(* Logix 5000 project; controller NSH_PLC1 vendor 1 type 14 code 167 rev 32.11; software revision 32.02; part 6 of 12 *)
(* tags used below, declared in another part *)
   HS_AlarmPulseHorn : BOOL;   // Huller Sheller, New Alarm, Pulse Horn
   HS_FaultResetHorn : BOOL;   // Hullwe Sheller, Fault Reset, sound Horn
   Num_Faults : DINT;   // Number of Huller-Sheller Faults
   Num_Warnings : DINT;   // Number of Huller-Sheller Warnings
   TempMotor : Motor;   // Temp Motor Tag for Subroutines
   BH1 : Motor;   // Auger
   BH1A : Motor;   // Fan
   BH1B : Motor;   // Rev.Fan
   BH1C : Motor;   // Rev. Arm
   BH1D : Motor;   // Airlock
   BH2 : Motor;   // S. Ele
   BH2A : Motor;   // Fan
   BH2B : Motor;   // Rev.Fan
   BH2C : Motor;   // Rev. Arm
   BH2D : Motor;   // Airlock
   BH3A : Motor;   // Fan
   BH3B : Motor;   // Rev.Fan
   BH3C : Motor;   // Rev. Arm
   BH3D : Motor;   // Airlock
   C1A : Motor;   // Auger
   C1B : Motor;   // Auger
   C2 : Motor;   // Auger
   C3A : Motor;   // Auger
   C3B : Motor;   // Auger
   C4 : Motor;   // Ele.
   C7 : Motor;   // Ele
   CR_LastBH1Fan : BOOL;   // Last Motor in Baghouse 1 Fans Running
   CR_RunBH_Fans : BOOL;   // Run Baghouse's Fans Relay
   CR_RunBH_FansCO : BOOL;   // Run Baghouse's Cleanout Relay
   CR_RunHS : BOOL;   // Run Hullers & Shellers Relay
   CR_RunPC1_Fans : BOOL;   // Pre Clean Run Line 1 Fans Relay
   CR_StopHS : BOOL;   // Stop Hullers & Shellers Relay
   D10 : Motor;   // Ele
   D1A : Motor;   // Auger
   D1B : Motor;   // Auger
   D2 : Motor;   // Auger
   D4 : Motor;   // Auger
   D5 : Motor;   // Auger
   D6 : Motor;   // Auger
   H1 : Motor;   // Conv.
   H11 : Motor;   // Ele.
   H12 : Motor;   // Auger
   H13 : Motor;   // Auger
   H14A : Motor;   // Shr. Roll
   H14B : Motor;   // Shr. Roll
   H14C : Motor;   // Vib.
   H16 : Motor;   // Auger
   H17 : Motor;   // Roll Fd.
   H18A : Motor;   // Shr. Roll
   H18B : Motor;   // Shr. Roll
   H18C : Motor;   // Vib.
   H19A : Motor;   // Aspirator
   H19B : Motor;   // Aspirator
   H22 : Motor;   // BMM
   H23A : Motor;   // Aspirator
   H23B : Motor;   // Aspirator
   H24A : Motor;   // Aspirator
   H24B : Motor;   // Aspirator
   H3A : Motor;   // Incline
   H3B : Motor;   // Ele.
   H4 : Motor;   // Auger
   H5 : Motor;   // Auger
   H6 : Motor;   // Roll Fd.
   H7 : Motor;   // BMM
   H8A : Motor;   // Aspirator
   H8B : Motor;   // Aspirator
   H9A : Motor;   // Aspirator
   H9B : Motor;   // Aspirator
   HS_Horn : BOOL;   // Huller Sheller, Horn Output
   HS_LastMotor : BOOL;   // Last Motor in Huller Sheller Sequence is Running
   HS_Starting : BOOL;   // Sheller Sequence is Starting, Prevent Preclean from Starting
   M12aA : Motor;   // Grav.Sep
   M12aB : Motor;   // Syntron
   M13aA : Motor;   // Grav.Sep
   M13aB : Motor;   // Syntron
   M14 : Motor;   // Vib.
   M15 : Motor;   // Ele.
   M16R : Motor;   // Conveyor
   M20 : Motor;   // Ele.
   M21 : Motor;   // Nolin
   M25 : Motor;   // Accept Vib.
   M33 : Motor;   // Belt
   M34 : Motor;   // Destoner
   M35 : Motor;   // Ele.
   M36A : Motor;   // G. Sep.
   M36B : Motor;   // R. Feeder.
   M42C : Motor;   // 3C Deck
   M42D : Motor;   // 3C Deck
   M43CA : Motor;   // Asp.
   M43CB : Motor;   // Asp.
   M43DA : Motor;   // Asp.
   M43DB : Motor;   // Asp.
   P2B : Motor;   // Stick Reel
   PB_HS_Inshell : BOOL;   // Hullers & Shellers Run Inshell Button
   PB_HS_Meats : BOOL;   // Hullers & Shellers Run Meats Button
   PB_StartHS : BOOL;   // Start Hullers & Shellers Button
   PB_StartPC1_Fans : BOOL;   // Pre Clean Start Line 1 Fans Button
   PB_StopHS : BOOL;   // Stop Hullers & Shellers Button
   PBB1D : Motor;   // Fan,
   PBL_HS_Inshell : BOOL;   // Hullers & Shellers Run Inshell Button Light
   PBL_HS_Meats : BOOL;   // Hullers & Shellers Run Meats Button Light
   PBL_StartHS : BOOL;   // Start Hullers & Shellers Button Light
   PBL_StopHS : BOOL;   // Stop Hullers & Shellers Button Light
   PC_FansStarting : BOOL;   // Pre Clean Fans Starting
   PC_LinesStarting : BOOL;   // Pre Clean Line 1 or 2 Starting
   PC_NoEstops : BOOL;   // PreClean, No Estops
   S11 : Motor;   // Ele.
   S12 : Motor;   // Auger
   T1 : Motor;   // Belt
   T2 : Motor;   // Belt
   T3 : Motor;   // Belt
   TMR_StartBH_Fans : TIMER;   // Start Baghouse's Fans Timer
   TMR_StartBH_FansCO : TIMER;   // Start Baghouse's Cleanout Timer
   TMR_StartHS : TIMER;   // Run Hullers & Shellers Warning Timer
(* HullerSheller, continued *)

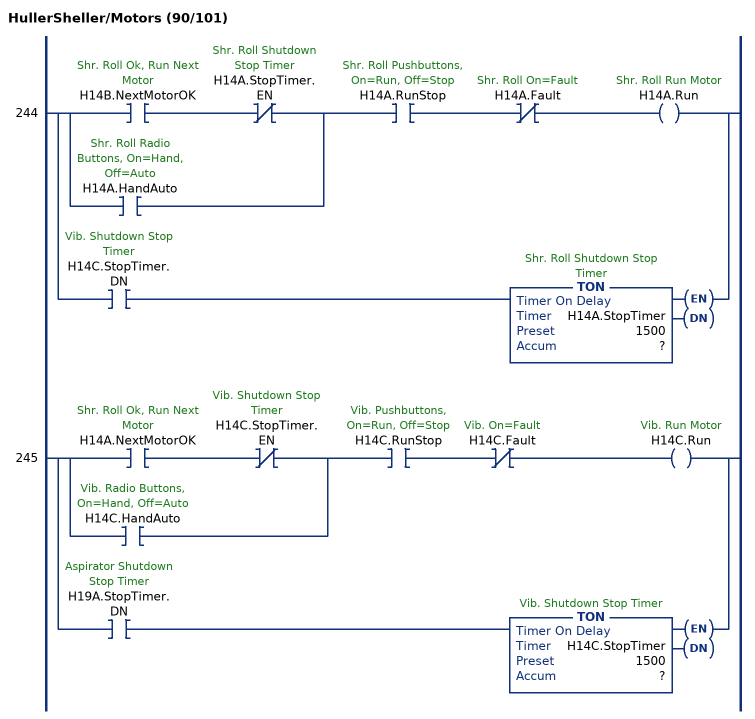
   244: [[XIC(H14B.NextMotorOK) XIO(H14A.StopTimer.EN) ,XIC(H14A.HandAuto) ] XIC(H14A.RunStop) XIO(H14A.Fault) OTE(H14A.Run) ,XIC(H14C.StopTimer.DN) TON(H14A.StopTimer,?,?) ];
   245: [[XIC(H14A.NextMotorOK) XIO(H14C.StopTimer.EN) ,XIC(H14C.HandAuto) ] XIC(H14C.RunStop) XIO(H14C.Fault) OTE(H14C.Run) ,XIC(H19A.StopTimer.DN) TON(H14C.StopTimer,?,?) ];
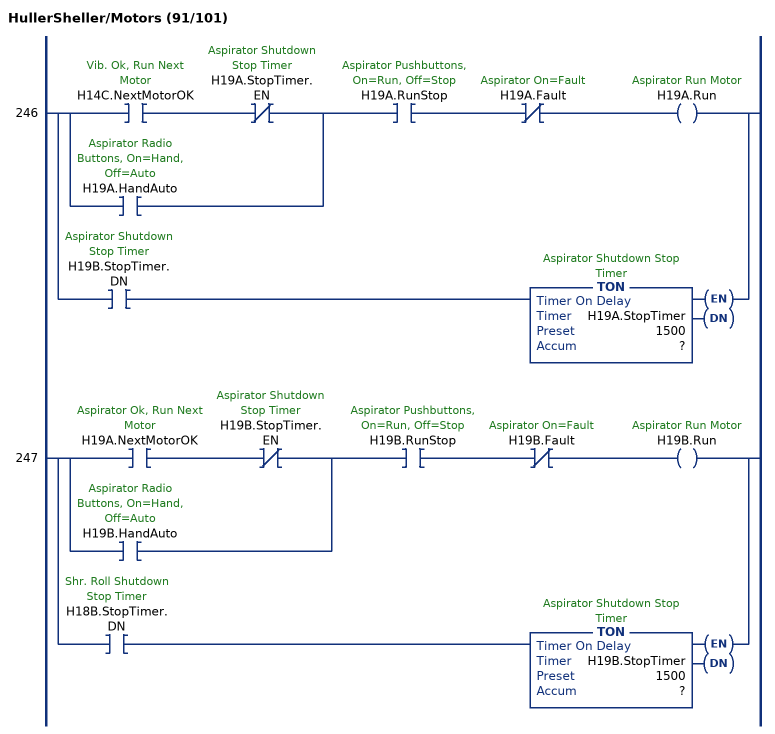
   246: [[XIC(H14C.NextMotorOK) XIO(H19A.StopTimer.EN) ,XIC(H19A.HandAuto) ] XIC(H19A.RunStop) XIO(H19A.Fault) OTE(H19A.Run) ,XIC(H19B.StopTimer.DN) TON(H19A.StopTimer,?,?) ];
   247: [[XIC(H19A.NextMotorOK) XIO(H19B.StopTimer.EN) ,XIC(H19B.HandAuto) ] XIC(H19B.RunStop) XIO(H19B.Fault) OTE(H19B.Run) ,XIC(H18B.StopTimer.DN) TON(H19B.StopTimer,?,?) ];
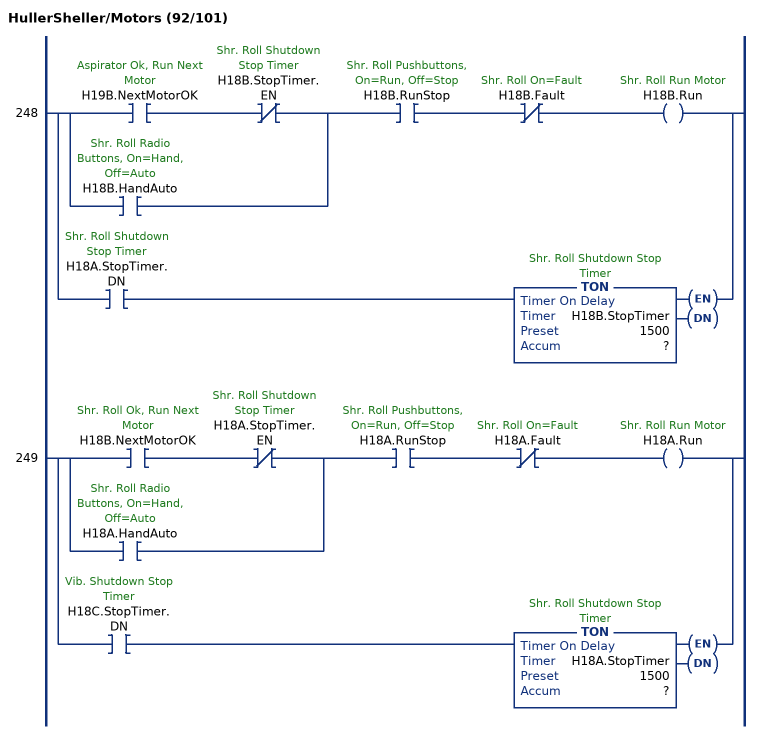
   248: [[XIC(H19B.NextMotorOK) XIO(H18B.StopTimer.EN) ,XIC(H18B.HandAuto) ] XIC(H18B.RunStop) XIO(H18B.Fault) OTE(H18B.Run) ,XIC(H18A.StopTimer.DN) TON(H18B.StopTimer,?,?) ];
   249: [[XIC(H18B.NextMotorOK) XIO(H18A.StopTimer.EN) ,XIC(H18A.HandAuto) ] XIC(H18A.RunStop) XIO(H18A.Fault) OTE(H18A.Run) ,XIC(H18C.StopTimer.DN) TON(H18A.StopTimer,?,?) ];
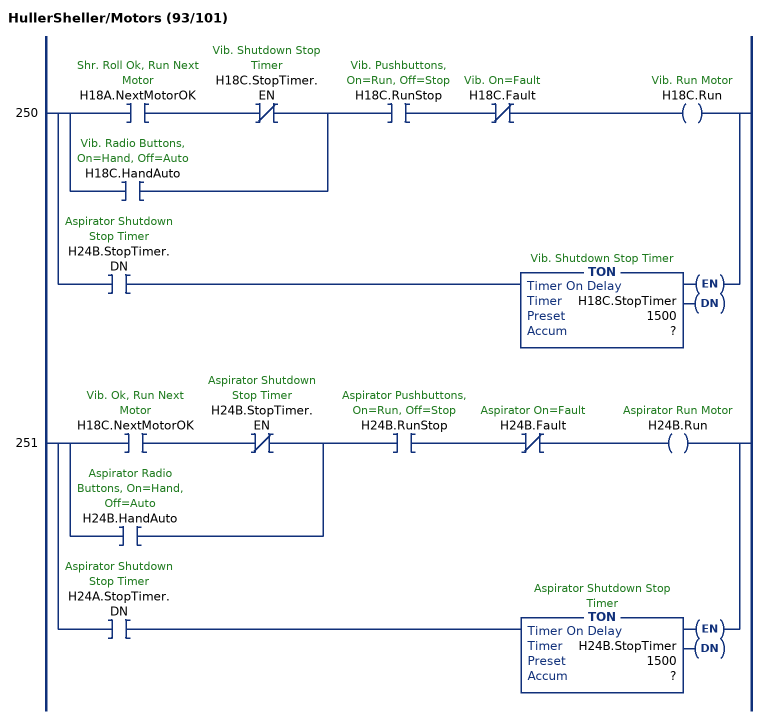
   250: [[XIC(H18A.NextMotorOK) XIO(H18C.StopTimer.EN) ,XIC(H18C.HandAuto) ] XIC(H18C.RunStop) XIO(H18C.Fault) OTE(H18C.Run) ,XIC(H24B.StopTimer.DN) TON(H18C.StopTimer,?,?) ];
   251: [[XIC(H18C.NextMotorOK) XIO(H24B.StopTimer.EN) ,XIC(H24B.HandAuto) ] XIC(H24B.RunStop) XIO(H24B.Fault) OTE(H24B.Run) ,XIC(H24A.StopTimer.DN) TON(H24B.StopTimer,?,?) ];
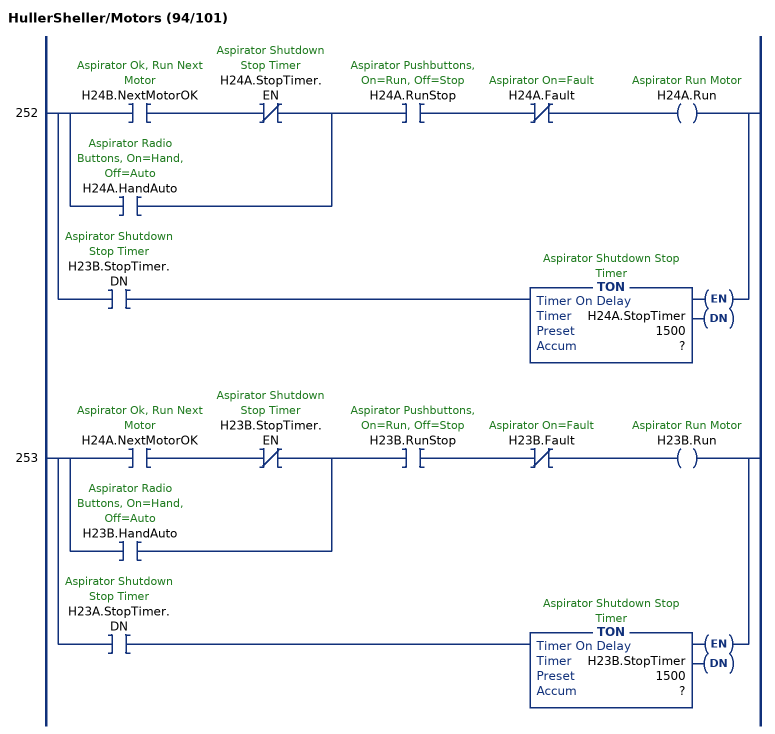
   252: [[XIC(H24B.NextMotorOK) XIO(H24A.StopTimer.EN) ,XIC(H24A.HandAuto) ] XIC(H24A.RunStop) XIO(H24A.Fault) OTE(H24A.Run) ,XIC(H23B.StopTimer.DN) TON(H24A.StopTimer,?,?) ];
   253: [[XIC(H24A.NextMotorOK) XIO(H23B.StopTimer.EN) ,XIC(H23B.HandAuto) ] XIC(H23B.RunStop) XIO(H23B.Fault) OTE(H23B.Run) ,XIC(H23A.StopTimer.DN) TON(H23B.StopTimer,?,?) ];
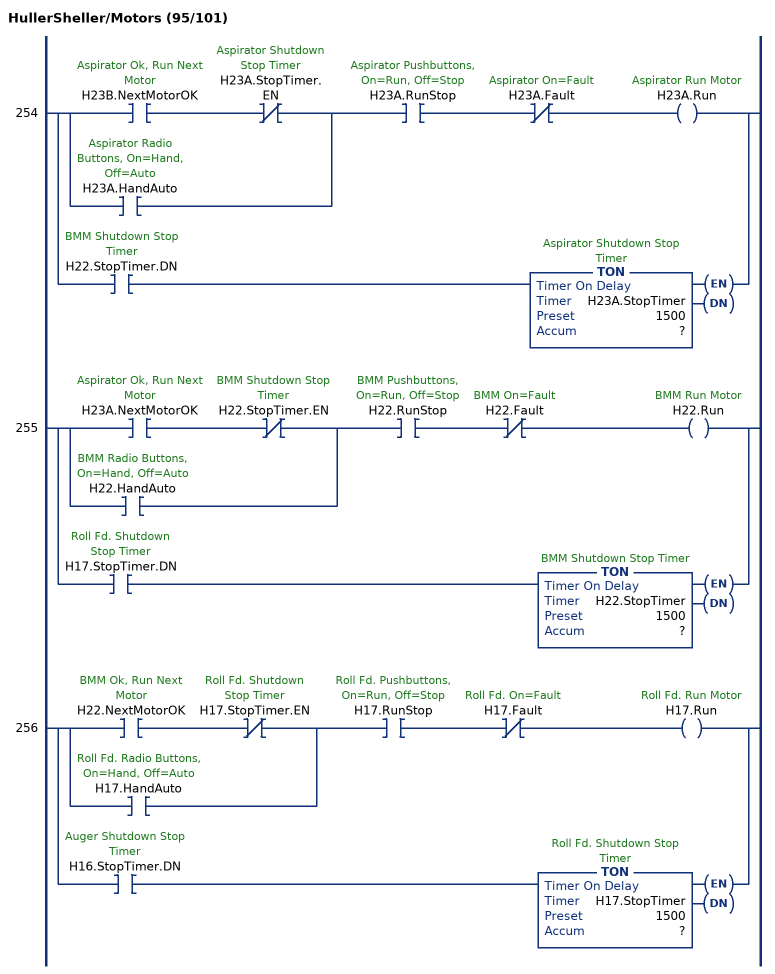
   254: [[XIC(H23B.NextMotorOK) XIO(H23A.StopTimer.EN) ,XIC(H23A.HandAuto) ] XIC(H23A.RunStop) XIO(H23A.Fault) OTE(H23A.Run) ,XIC(H22.StopTimer.DN) TON(H23A.StopTimer,?,?) ];
   255: [[XIC(H23A.NextMotorOK) XIO(H22.StopTimer.EN) ,XIC(H22.HandAuto) ] XIC(H22.RunStop) XIO(H22.Fault) OTE(H22.Run) ,XIC(H17.StopTimer.DN) TON(H22.StopTimer,?,?) ];
   256: [[XIC(H22.NextMotorOK) XIO(H17.StopTimer.EN) ,XIC(H17.HandAuto) ] XIC(H17.RunStop) XIO(H17.Fault) OTE(H17.Run) ,XIC(H16.StopTimer.DN) TON(H17.StopTimer,?,?) ];
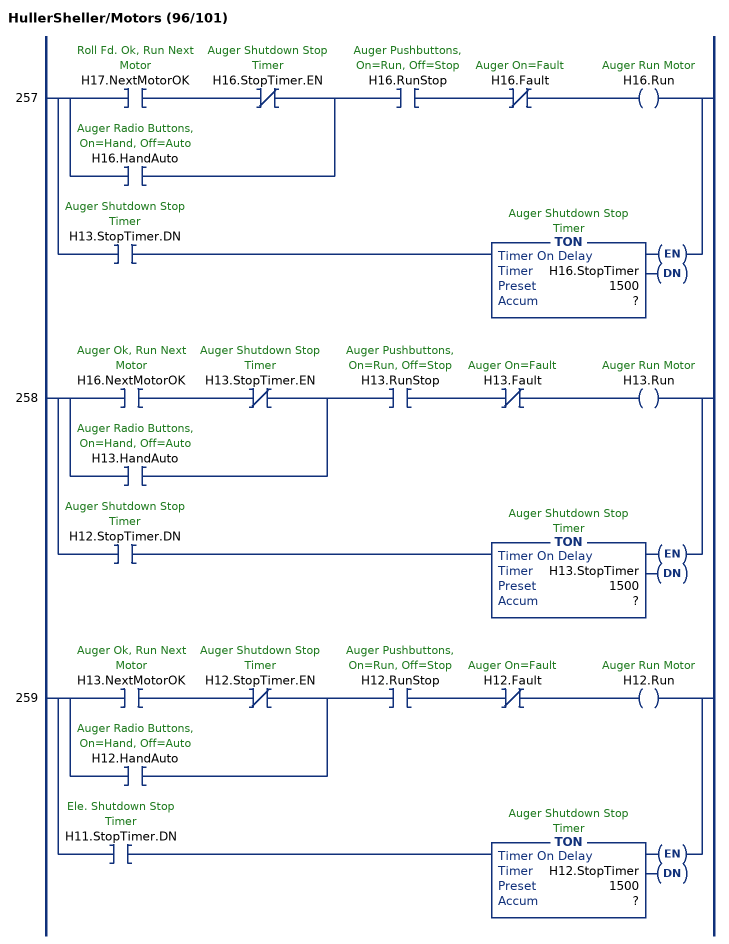
   257: [[XIC(H17.NextMotorOK) XIO(H16.StopTimer.EN) ,XIC(H16.HandAuto) ] XIC(H16.RunStop) XIO(H16.Fault) OTE(H16.Run) ,XIC(H13.StopTimer.DN) TON(H16.StopTimer,?,?) ];
   258: [[XIC(H16.NextMotorOK) XIO(H13.StopTimer.EN) ,XIC(H13.HandAuto) ] XIC(H13.RunStop) XIO(H13.Fault) OTE(H13.Run) ,XIC(H12.StopTimer.DN) TON(H13.StopTimer,?,?) ];
   259: [[XIC(H13.NextMotorOK) XIO(H12.StopTimer.EN) ,XIC(H12.HandAuto) ] XIC(H12.RunStop) XIO(H12.Fault) OTE(H12.Run) ,XIC(H11.StopTimer.DN) TON(H12.StopTimer,?,?) ];
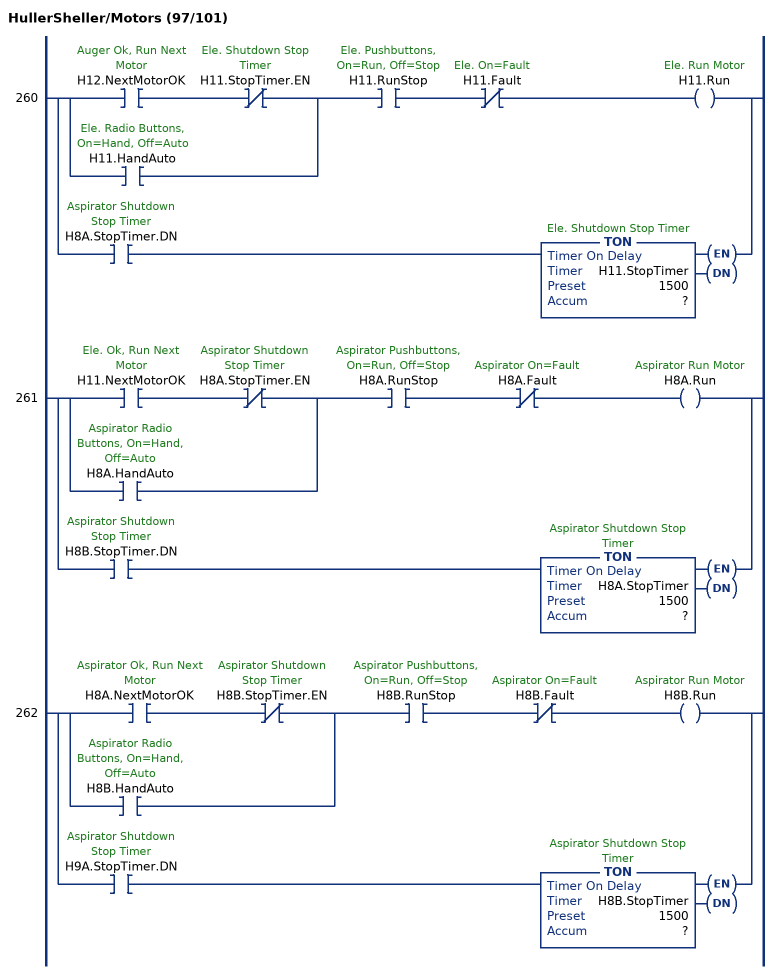
   260: [[XIC(H12.NextMotorOK) XIO(H11.StopTimer.EN) ,XIC(H11.HandAuto) ] XIC(H11.RunStop) XIO(H11.Fault) OTE(H11.Run) ,XIC(H8A.StopTimer.DN) TON(H11.StopTimer,?,?) ];
   261: [[XIC(H11.NextMotorOK) XIO(H8A.StopTimer.EN) ,XIC(H8A.HandAuto) ] XIC(H8A.RunStop) XIO(H8A.Fault) OTE(H8A.Run) ,XIC(H8B.StopTimer.DN) TON(H8A.StopTimer,?,?) ];
   262: [[XIC(H8A.NextMotorOK) XIO(H8B.StopTimer.EN) ,XIC(H8B.HandAuto) ] XIC(H8B.RunStop) XIO(H8B.Fault) OTE(H8B.Run) ,XIC(H9A.StopTimer.DN) TON(H8B.StopTimer,?,?) ];
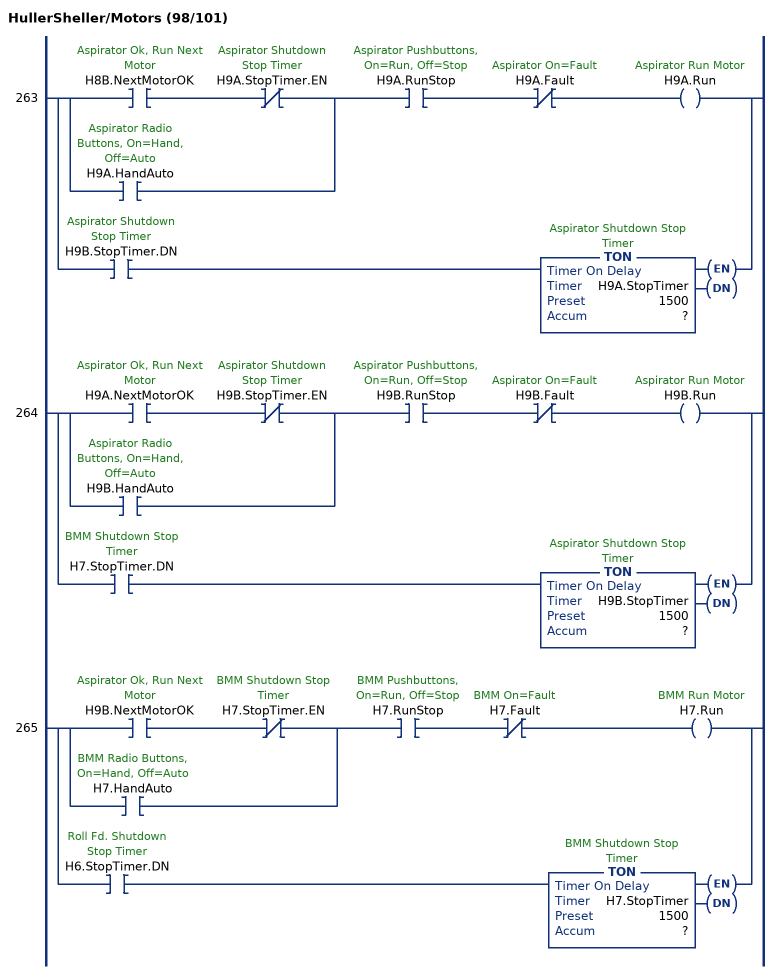
   263: [[XIC(H8B.NextMotorOK) XIO(H9A.StopTimer.EN) ,XIC(H9A.HandAuto) ] XIC(H9A.RunStop) XIO(H9A.Fault) OTE(H9A.Run) ,XIC(H9B.StopTimer.DN) TON(H9A.StopTimer,?,?) ];
   264: [[XIC(H9A.NextMotorOK) XIO(H9B.StopTimer.EN) ,XIC(H9B.HandAuto) ] XIC(H9B.RunStop) XIO(H9B.Fault) OTE(H9B.Run) ,XIC(H7.StopTimer.DN) TON(H9B.StopTimer,?,?) ];
   265: [[XIC(H9B.NextMotorOK) XIO(H7.StopTimer.EN) ,XIC(H7.HandAuto) ] XIC(H7.RunStop) XIO(H7.Fault) OTE(H7.Run) ,XIC(H6.StopTimer.DN) TON(H7.StopTimer,?,?) ];
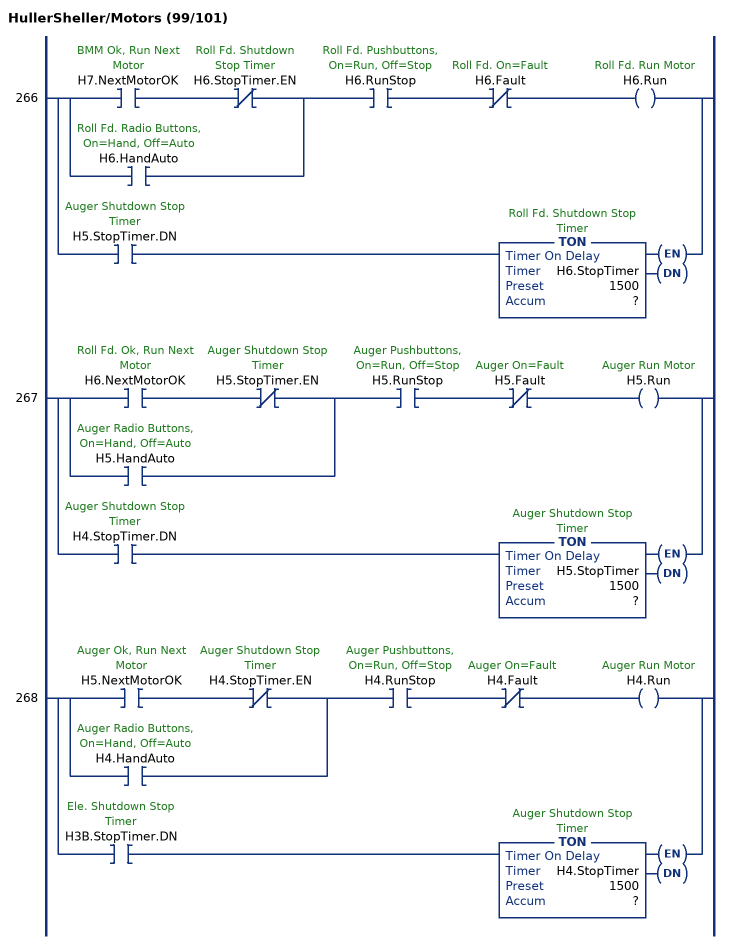
   266: [[XIC(H7.NextMotorOK) XIO(H6.StopTimer.EN) ,XIC(H6.HandAuto) ] XIC(H6.RunStop) XIO(H6.Fault) OTE(H6.Run) ,XIC(H5.StopTimer.DN) TON(H6.StopTimer,?,?) ];
   267: [[XIC(H6.NextMotorOK) XIO(H5.StopTimer.EN) ,XIC(H5.HandAuto) ] XIC(H5.RunStop) XIO(H5.Fault) OTE(H5.Run) ,XIC(H4.StopTimer.DN) TON(H5.StopTimer,?,?) ];
   268: [[XIC(H5.NextMotorOK) XIO(H4.StopTimer.EN) ,XIC(H4.HandAuto) ] XIC(H4.RunStop) XIO(H4.Fault) OTE(H4.Run) ,XIC(H3B.StopTimer.DN) TON(H4.StopTimer,?,?) ];
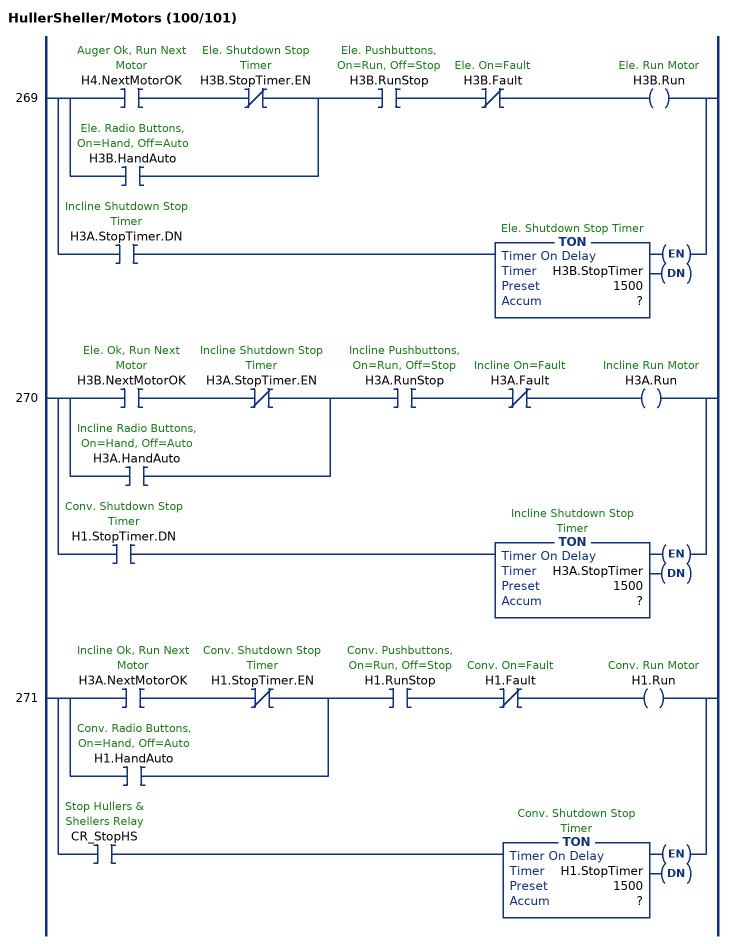
   269: [[XIC(H4.NextMotorOK) XIO(H3B.StopTimer.EN) ,XIC(H3B.HandAuto) ] XIC(H3B.RunStop) XIO(H3B.Fault) OTE(H3B.Run) ,XIC(H3A.StopTimer.DN) TON(H3B.StopTimer,?,?) ];
   270: [[XIC(H3B.NextMotorOK) XIO(H3A.StopTimer.EN) ,XIC(H3A.HandAuto) ] XIC(H3A.RunStop) XIO(H3A.Fault) OTE(H3A.Run) ,XIC(H1.StopTimer.DN) TON(H3A.StopTimer,?,?) ];
   271: [[XIC(H3A.NextMotorOK) XIO(H1.StopTimer.EN) ,XIC(H1.HandAuto) ] XIC(H1.RunStop) XIO(H1.Fault) OTE(H1.Run) ,XIC(CR_StopHS) TON(H1.StopTimer,?,?) ];
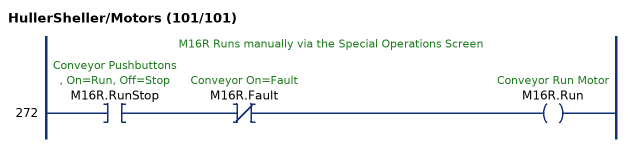
   // M16R Runs manually via the Special Operations Screen
   272: XIC(M16R.RunStop)XIO(M16R.Fault)OTE(M16R.Run);
END_ROUTINE

ROUTINE MotorStatusSUB   (* ladder *)
// Update Status Subroutine
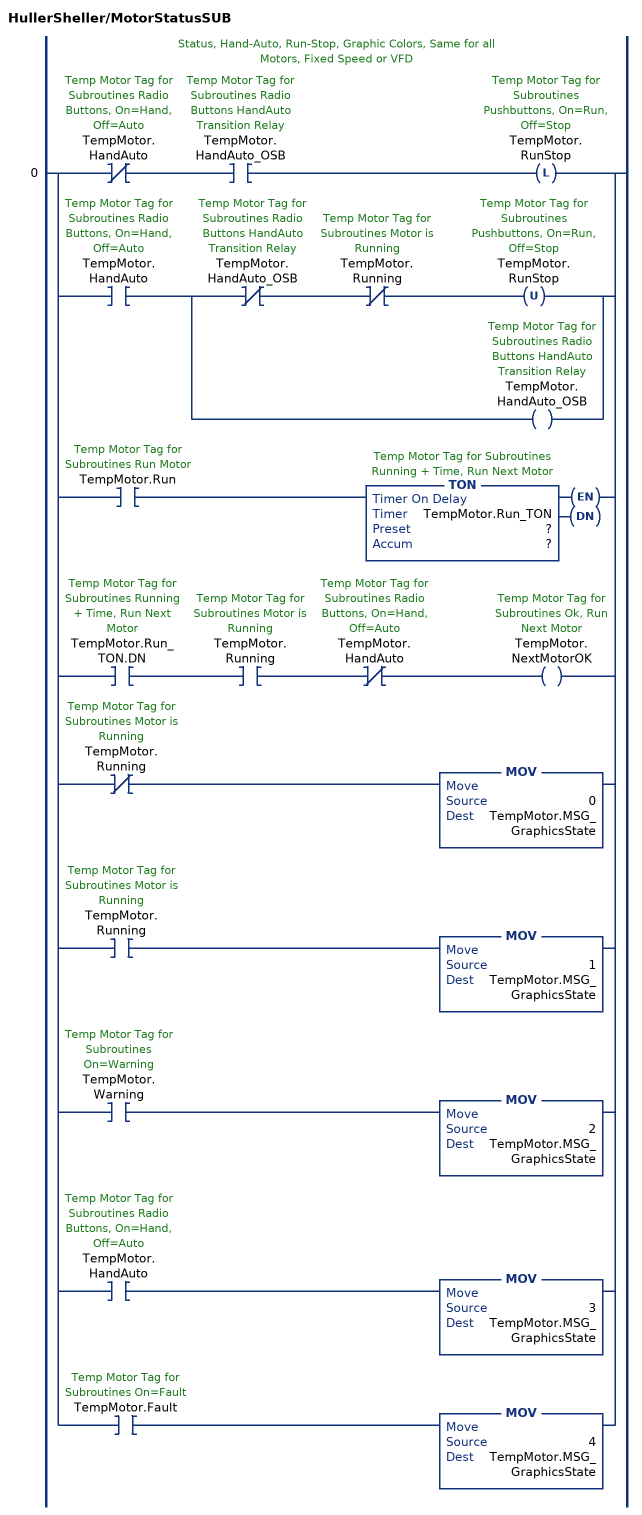
   // Status, Hand-Auto, Run-Stop, Graphic Colors, Same for all
   // Motors, Fixed Speed or VFD
   0: [XIO(TempMotor.HandAuto) XIC(TempMotor.HandAuto_OSB) OTL(TempMotor.RunStop) ,XIC(TempMotor.HandAuto) [XIO(TempMotor.HandAuto_OSB) XIO(TempMotor.Running) OTU(TempMotor.RunStop) ,OTE(TempMotor.HandAuto_OSB) ] ,XIC(TempMotor.Run) TON(TempMotor.Run_TON,?,?) ,XIC(TempMotor.Run_TON.DN) XIC(TempMotor.Running) XIO(TempMotor.HandAuto) OTE(TempMotor.NextMotorOK) ,XIO(TempMotor.Running) MOV(0,TempMotor.MSG_GraphicsState) ,XIC(TempMotor.Running) MOV(1,TempMotor.MSG_GraphicsState) ,XIC(TempMotor.Warning) MOV(2,TempMotor.MSG_GraphicsState) ,XIC(TempMotor.HandAuto) MOV(3,TempMotor.MSG_GraphicsState) ,XIC(TempMotor.Fault) MOV(4,TempMotor.MSG_GraphicsState) ];
END_ROUTINE

ROUTINE StartStopMCRs   (* ladder *)
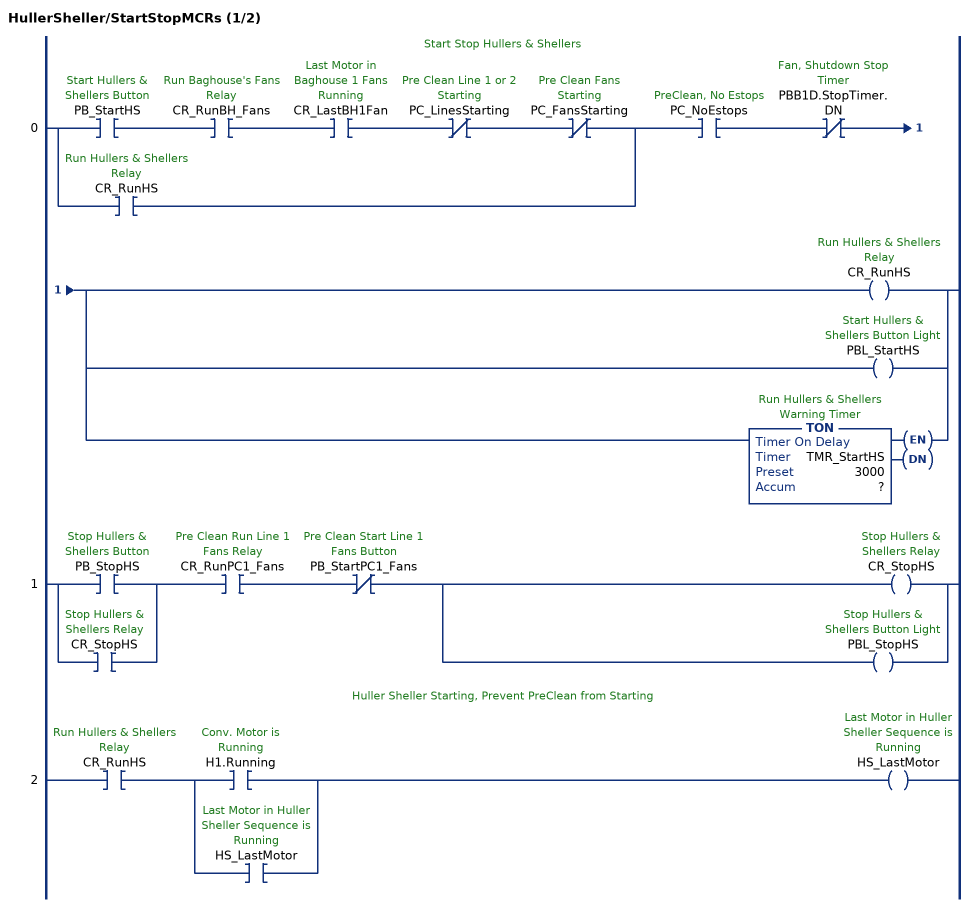
   // Start Stop Hullers & Shellers
   0: [XIC(PB_StartHS) XIC(CR_RunBH_Fans) XIC(CR_LastBH1Fan) XIO(PC_LinesStarting) XIO(PC_FansStarting) ,XIC(CR_RunHS) ]XIC(PC_NoEstops)XIO(PBB1D.StopTimer.DN)[OTE(CR_RunHS) ,OTE(PBL_StartHS) ,TON(TMR_StartHS,?,?) ];
   1: [XIC(PB_StopHS) ,XIC(CR_StopHS) ]XIC(CR_RunPC1_Fans)XIO(PB_StartPC1_Fans)[OTE(CR_StopHS) ,OTE(PBL_StopHS) ];
   // Huller Sheller Starting, Prevent PreClean from Starting
   2: XIC(CR_RunHS)[XIC(H1.Running) ,XIC(HS_LastMotor) ]OTE(HS_LastMotor);
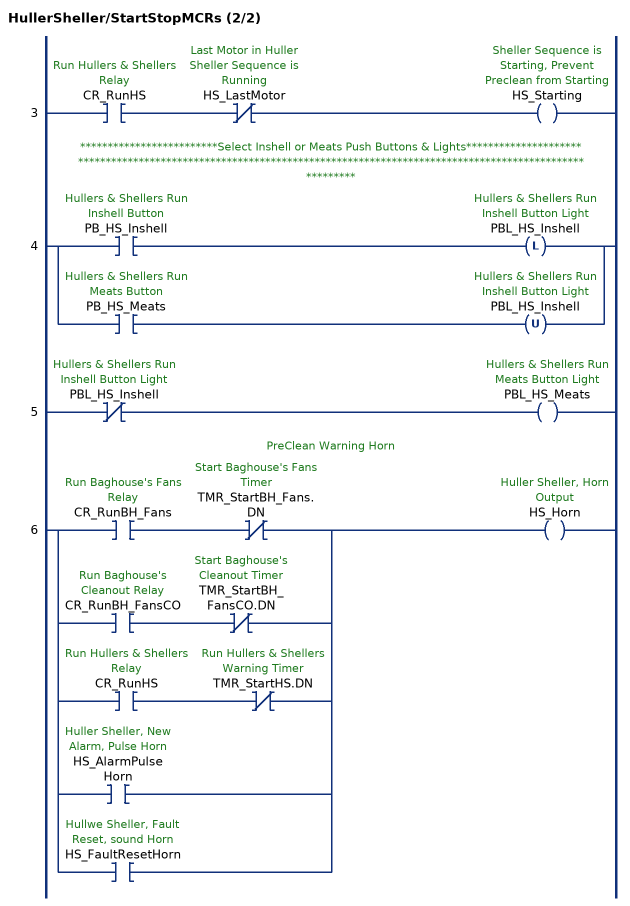
   3: XIC(CR_RunHS)XIO(HS_LastMotor)OTE(HS_Starting);
   // *************************Select Inshell or Meats Push Buttons & Lights*********************
   // *****************************************************************************************************
   4: [XIC(PB_HS_Inshell) OTL(PBL_HS_Inshell) ,XIC(PB_HS_Meats) OTU(PBL_HS_Inshell) ];
   5: XIO(PBL_HS_Inshell)OTE(PBL_HS_Meats);
   // PreClean Warning Horn
   6: [XIC(CR_RunBH_Fans) XIO(TMR_StartBH_Fans.DN) ,XIC(CR_RunBH_FansCO) XIO(TMR_StartBH_FansCO.DN) ,XIC(CR_RunHS) XIO(TMR_StartHS.DN) ,XIC(HS_AlarmPulseHorn) ,XIC(HS_FaultResetHorn) ]OTE(HS_Horn);
END_ROUTINE

ROUTINE StatusAlarms   (* ladder *)
// Motor Status And Alarms
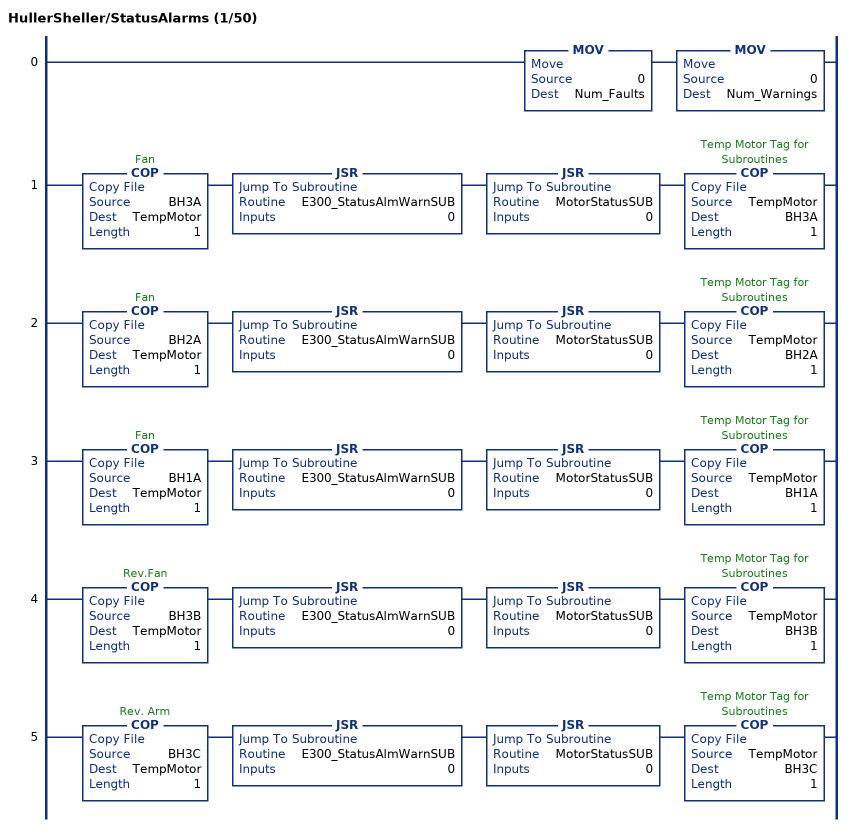
   0: MOV(0,Num_Faults)MOV(0,Num_Warnings);
   1: COP(BH3A,TempMotor,1)JSR(E300_StatusAlmWarnSUB,0)JSR(MotorStatusSUB,0)COP(TempMotor,BH3A,1);
   2: COP(BH2A,TempMotor,1)JSR(E300_StatusAlmWarnSUB,0)JSR(MotorStatusSUB,0)COP(TempMotor,BH2A,1);
   3: COP(BH1A,TempMotor,1)JSR(E300_StatusAlmWarnSUB,0)JSR(MotorStatusSUB,0)COP(TempMotor,BH1A,1);
   4: COP(BH3B,TempMotor,1)JSR(E300_StatusAlmWarnSUB,0)JSR(MotorStatusSUB,0)COP(TempMotor,BH3B,1);
   5: COP(BH3C,TempMotor,1)JSR(E300_StatusAlmWarnSUB,0)JSR(MotorStatusSUB,0)COP(TempMotor,BH3C,1);
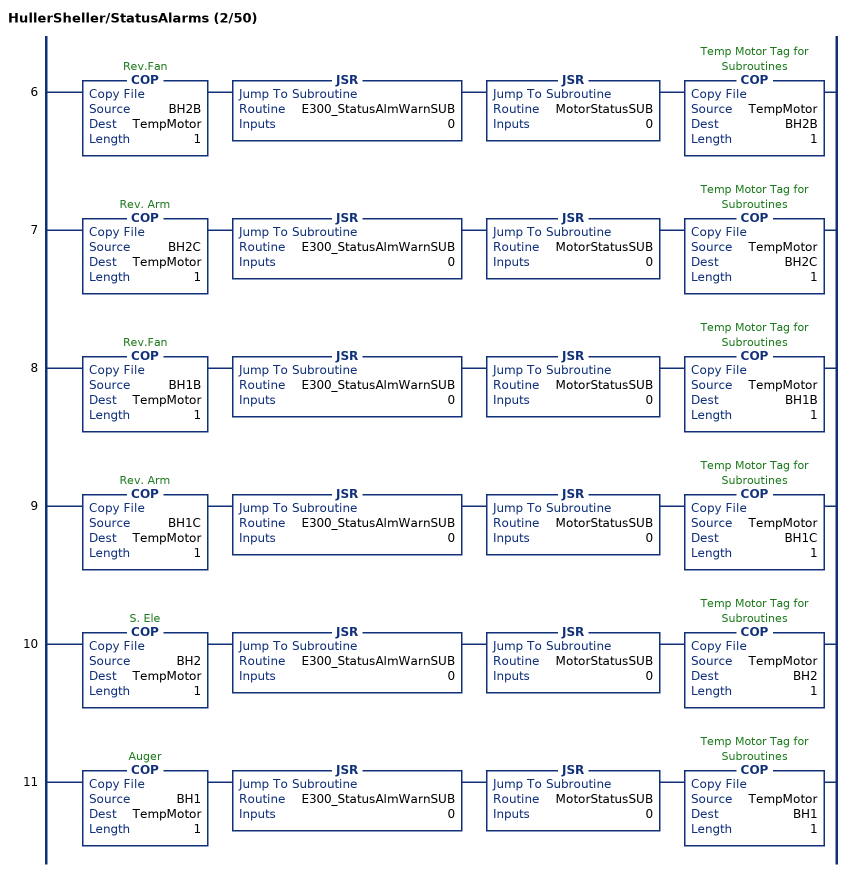
   6: COP(BH2B,TempMotor,1)JSR(E300_StatusAlmWarnSUB,0)JSR(MotorStatusSUB,0)COP(TempMotor,BH2B,1);
   7: COP(BH2C,TempMotor,1)JSR(E300_StatusAlmWarnSUB,0)JSR(MotorStatusSUB,0)COP(TempMotor,BH2C,1);
   8: COP(BH1B,TempMotor,1)JSR(E300_StatusAlmWarnSUB,0)JSR(MotorStatusSUB,0)COP(TempMotor,BH1B,1);
   9: COP(BH1C,TempMotor,1)JSR(E300_StatusAlmWarnSUB,0)JSR(MotorStatusSUB,0)COP(TempMotor,BH1C,1);
   10: COP(BH2,TempMotor,1)JSR(E300_StatusAlmWarnSUB,0)JSR(MotorStatusSUB,0)COP(TempMotor,BH2,1);
   11: COP(BH1,TempMotor,1)JSR(E300_StatusAlmWarnSUB,0)JSR(MotorStatusSUB,0)COP(TempMotor,BH1,1);
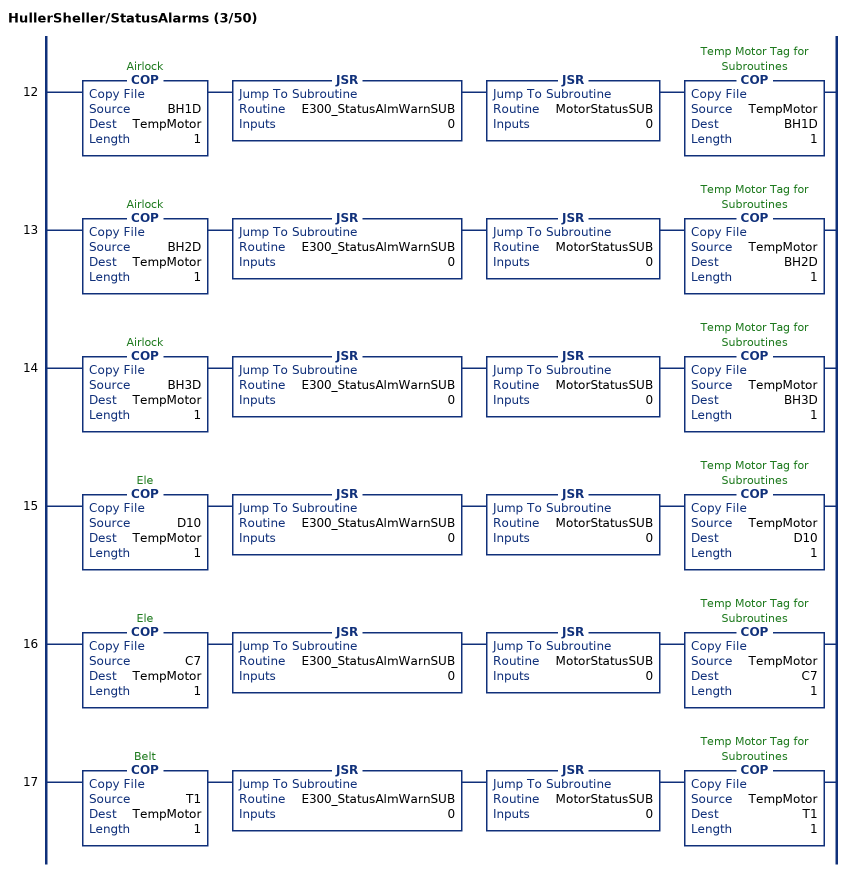
   12: COP(BH1D,TempMotor,1)JSR(E300_StatusAlmWarnSUB,0)JSR(MotorStatusSUB,0)COP(TempMotor,BH1D,1);
   13: COP(BH2D,TempMotor,1)JSR(E300_StatusAlmWarnSUB,0)JSR(MotorStatusSUB,0)COP(TempMotor,BH2D,1);
   14: COP(BH3D,TempMotor,1)JSR(E300_StatusAlmWarnSUB,0)JSR(MotorStatusSUB,0)COP(TempMotor,BH3D,1);
   15: COP(D10,TempMotor,1)JSR(E300_StatusAlmWarnSUB,0)JSR(MotorStatusSUB,0)COP(TempMotor,D10,1);
   16: COP(C7,TempMotor,1)JSR(E300_StatusAlmWarnSUB,0)JSR(MotorStatusSUB,0)COP(TempMotor,C7,1);
   17: COP(T1,TempMotor,1)JSR(E300_StatusAlmWarnSUB,0)JSR(MotorStatusSUB,0)COP(TempMotor,T1,1);
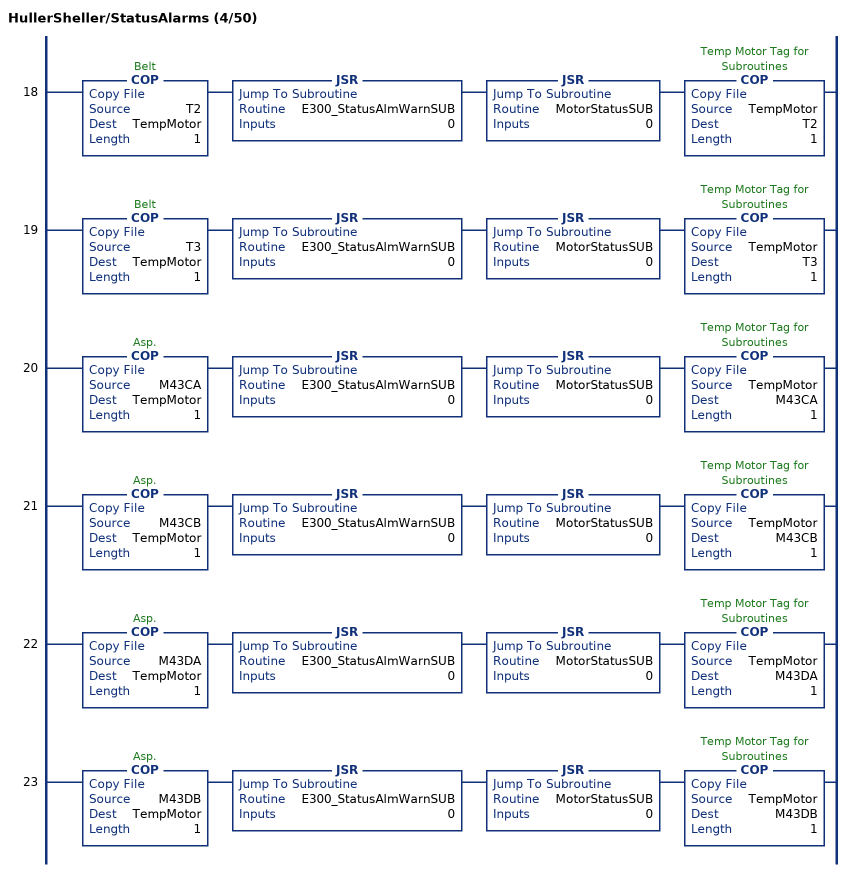
   18: COP(T2,TempMotor,1)JSR(E300_StatusAlmWarnSUB,0)JSR(MotorStatusSUB,0)COP(TempMotor,T2,1);
   19: COP(T3,TempMotor,1)JSR(E300_StatusAlmWarnSUB,0)JSR(MotorStatusSUB,0)COP(TempMotor,T3,1);
   20: COP(M43CA,TempMotor,1)JSR(E300_StatusAlmWarnSUB,0)JSR(MotorStatusSUB,0)COP(TempMotor,M43CA,1);
   21: COP(M43CB,TempMotor,1)JSR(E300_StatusAlmWarnSUB,0)JSR(MotorStatusSUB,0)COP(TempMotor,M43CB,1);
   22: COP(M43DA,TempMotor,1)JSR(E300_StatusAlmWarnSUB,0)JSR(MotorStatusSUB,0)COP(TempMotor,M43DA,1);
   23: COP(M43DB,TempMotor,1)JSR(E300_StatusAlmWarnSUB,0)JSR(MotorStatusSUB,0)COP(TempMotor,M43DB,1);
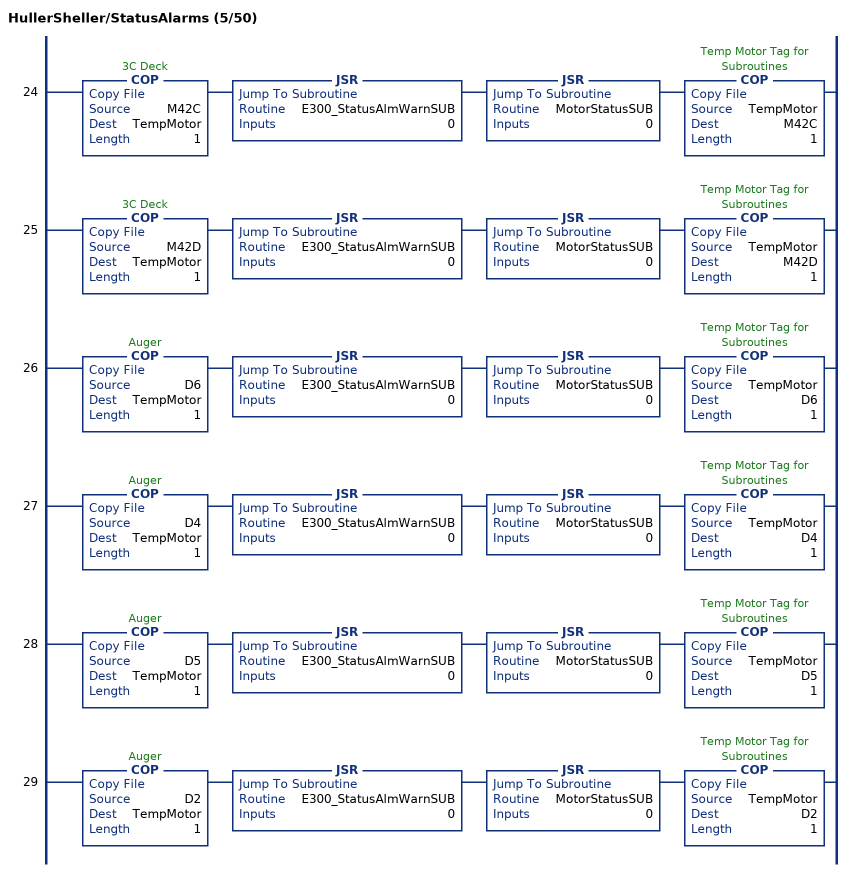
   24: COP(M42C,TempMotor,1)JSR(E300_StatusAlmWarnSUB,0)JSR(MotorStatusSUB,0)COP(TempMotor,M42C,1);
   25: COP(M42D,TempMotor,1)JSR(E300_StatusAlmWarnSUB,0)JSR(MotorStatusSUB,0)COP(TempMotor,M42D,1);
   26: COP(D6,TempMotor,1)JSR(E300_StatusAlmWarnSUB,0)JSR(MotorStatusSUB,0)COP(TempMotor,D6,1);
   27: COP(D4,TempMotor,1)JSR(E300_StatusAlmWarnSUB,0)JSR(MotorStatusSUB,0)COP(TempMotor,D4,1);
   28: COP(D5,TempMotor,1)JSR(E300_StatusAlmWarnSUB,0)JSR(MotorStatusSUB,0)COP(TempMotor,D5,1);
   29: COP(D2,TempMotor,1)JSR(E300_StatusAlmWarnSUB,0)JSR(MotorStatusSUB,0)COP(TempMotor,D2,1);
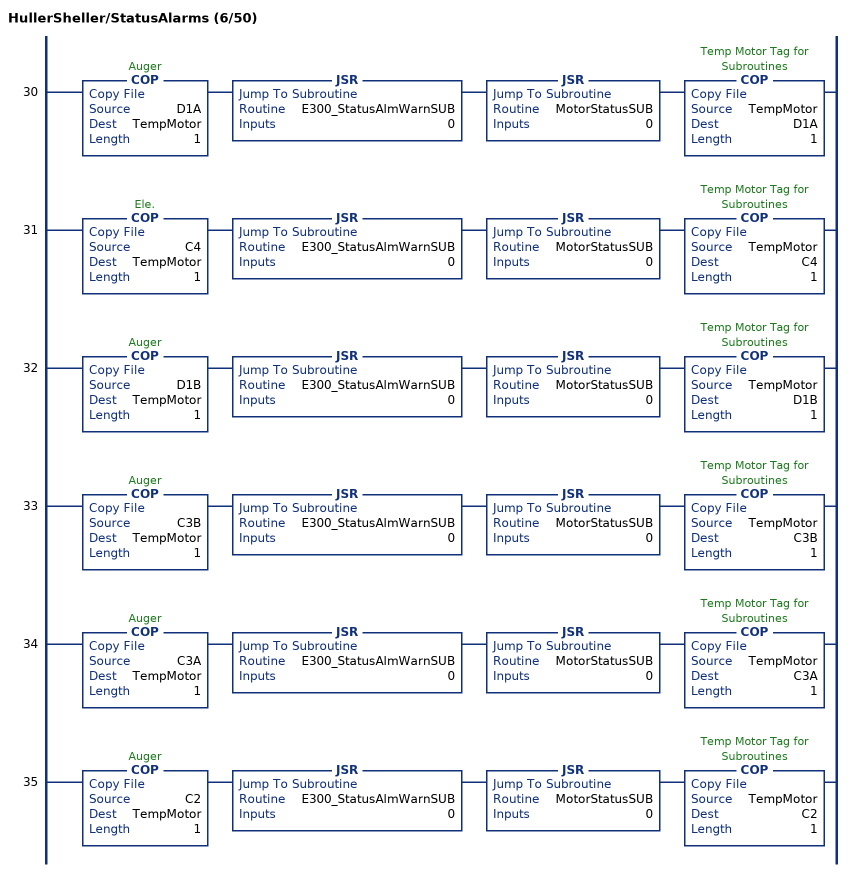
   30: COP(D1A,TempMotor,1)JSR(E300_StatusAlmWarnSUB,0)JSR(MotorStatusSUB,0)COP(TempMotor,D1A,1);
   31: COP(C4,TempMotor,1)JSR(E300_StatusAlmWarnSUB,0)JSR(MotorStatusSUB,0)COP(TempMotor,C4,1);
   32: COP(D1B,TempMotor,1)JSR(E300_StatusAlmWarnSUB,0)JSR(MotorStatusSUB,0)COP(TempMotor,D1B,1);
   33: COP(C3B,TempMotor,1)JSR(E300_StatusAlmWarnSUB,0)JSR(MotorStatusSUB,0)COP(TempMotor,C3B,1);
   34: COP(C3A,TempMotor,1)JSR(E300_StatusAlmWarnSUB,0)JSR(MotorStatusSUB,0)COP(TempMotor,C3A,1);
   35: COP(C2,TempMotor,1)JSR(E300_StatusAlmWarnSUB,0)JSR(MotorStatusSUB,0)COP(TempMotor,C2,1);
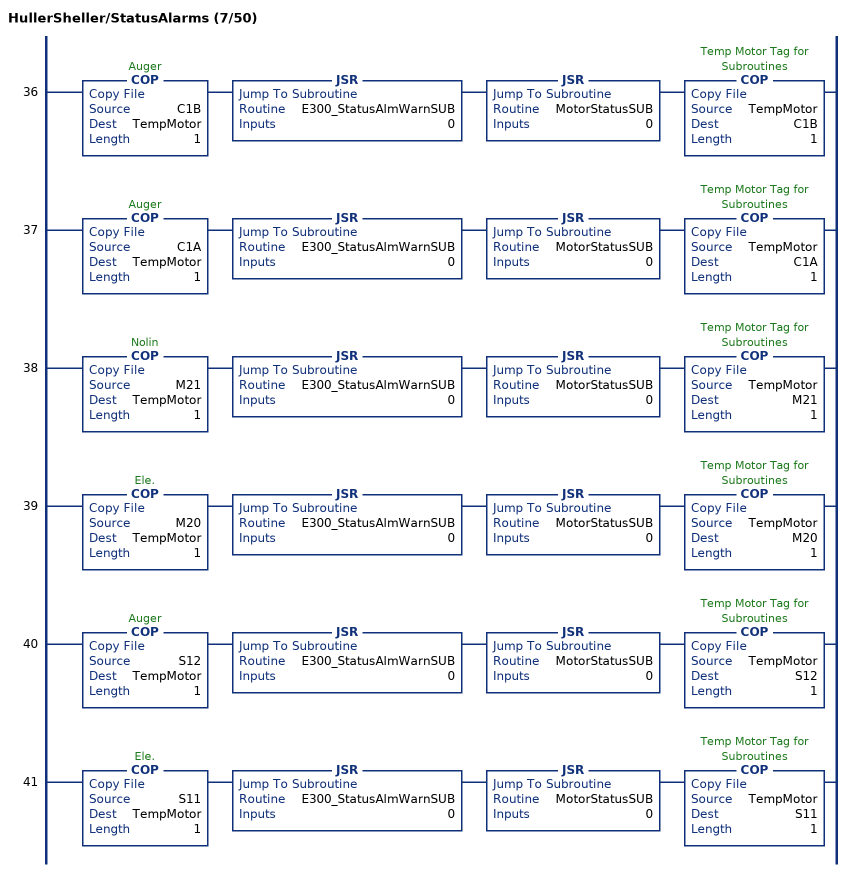
   36: COP(C1B,TempMotor,1)JSR(E300_StatusAlmWarnSUB,0)JSR(MotorStatusSUB,0)COP(TempMotor,C1B,1);
   37: COP(C1A,TempMotor,1)JSR(E300_StatusAlmWarnSUB,0)JSR(MotorStatusSUB,0)COP(TempMotor,C1A,1);
   38: COP(M21,TempMotor,1)JSR(E300_StatusAlmWarnSUB,0)JSR(MotorStatusSUB,0)COP(TempMotor,M21,1);
   39: COP(M20,TempMotor,1)JSR(E300_StatusAlmWarnSUB,0)JSR(MotorStatusSUB,0)COP(TempMotor,M20,1);
   40: COP(S12,TempMotor,1)JSR(E300_StatusAlmWarnSUB,0)JSR(MotorStatusSUB,0)COP(TempMotor,S12,1);
   41: COP(S11,TempMotor,1)JSR(E300_StatusAlmWarnSUB,0)JSR(MotorStatusSUB,0)COP(TempMotor,S11,1);
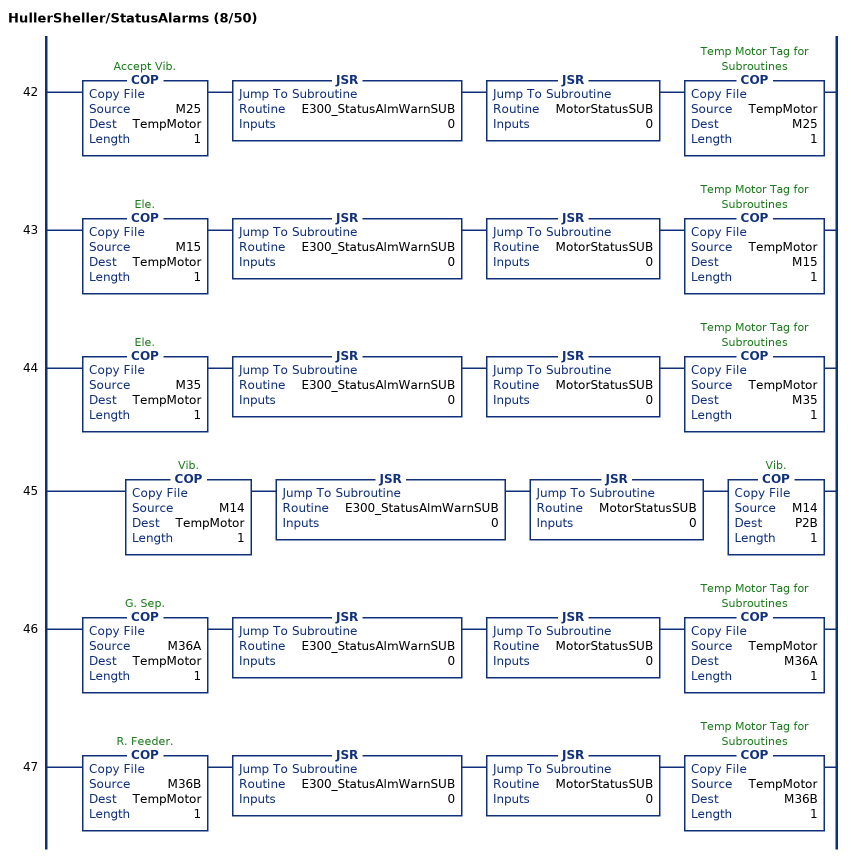
   42: COP(M25,TempMotor,1)JSR(E300_StatusAlmWarnSUB,0)JSR(MotorStatusSUB,0)COP(TempMotor,M25,1);
   43: COP(M15,TempMotor,1)JSR(E300_StatusAlmWarnSUB,0)JSR(MotorStatusSUB,0)COP(TempMotor,M15,1);
   44: COP(M35,TempMotor,1)JSR(E300_StatusAlmWarnSUB,0)JSR(MotorStatusSUB,0)COP(TempMotor,M35,1);
   45: COP(M14,TempMotor,1)JSR(E300_StatusAlmWarnSUB,0)JSR(MotorStatusSUB,0)COP(M14,P2B,1);
   46: COP(M36A,TempMotor,1)JSR(E300_StatusAlmWarnSUB,0)JSR(MotorStatusSUB,0)COP(TempMotor,M36A,1);
   47: COP(M36B,TempMotor,1)JSR(E300_StatusAlmWarnSUB,0)JSR(MotorStatusSUB,0)COP(TempMotor,M36B,1);
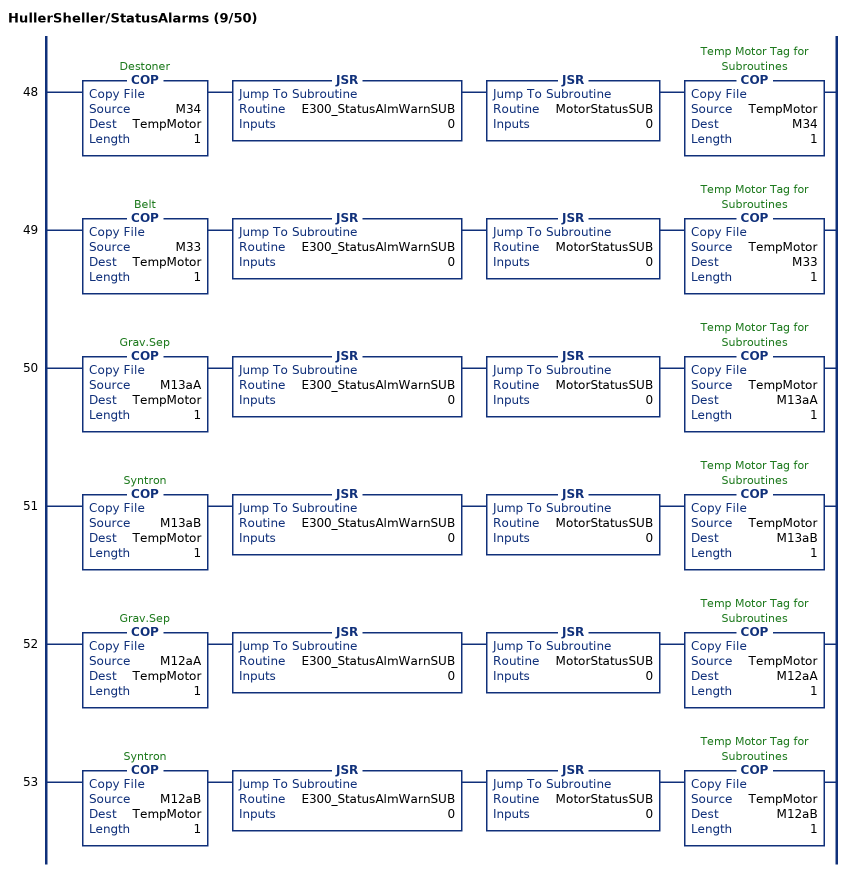
   48: COP(M34,TempMotor,1)JSR(E300_StatusAlmWarnSUB,0)JSR(MotorStatusSUB,0)COP(TempMotor,M34,1);
   49: COP(M33,TempMotor,1)JSR(E300_StatusAlmWarnSUB,0)JSR(MotorStatusSUB,0)COP(TempMotor,M33,1);
   50: COP(M13aA,TempMotor,1)JSR(E300_StatusAlmWarnSUB,0)JSR(MotorStatusSUB,0)COP(TempMotor,M13aA,1);
   51: COP(M13aB,TempMotor,1)JSR(E300_StatusAlmWarnSUB,0)JSR(MotorStatusSUB,0)COP(TempMotor,M13aB,1);
   52: COP(M12aA,TempMotor,1)JSR(E300_StatusAlmWarnSUB,0)JSR(MotorStatusSUB,0)COP(TempMotor,M12aA,1);
   53: COP(M12aB,TempMotor,1)JSR(E300_StatusAlmWarnSUB,0)JSR(MotorStatusSUB,0)COP(TempMotor,M12aB,1);
